{attribute 'GeneratedUsingTerminal: EL3773-0000-0021'}
{attribute addProperty BoxType "EL3773-0000-0021"}
{attribute addProperty Id "I1_SamplesAT %I*I1_Samples_2549228720"}
{attribute addProperty CRC "2663418686"}
{attribute addProperty Size "20"}
TYPE L1_Current_Samples_9EC08B3E EXTENDS TcoIo.InputBase_8311D824 :
STRUCT
    {attribute addProperty Name "I1_Samples"}
    I1_Samples AT %I* : I1_Samples_25492287;
END_STRUCT
END_TYPE

(* stored: Version 1.2.0.0, ProductVersion 3.1.4024.11
   DUT L1_Current_Samples_9EC08B3E: Id {ae572fe9-2171-076c-2704-a1dc2569e7fa} *)
